FUNCTION "ASCF_GetVDIntOutputList" : Word
{ S7_Optimized_Access := 'TRUE' }
VERSION : 0.1
   VAR_INPUT
      Index : UInt;
   END_VAR

   VAR_OUTPUT
      QC : Byte;
      Value : DInt;
   END_VAR

   VAR_IN_OUT
      Outputs : Array[*] of "ASCF_CL_OutputType";
   END_VAR

   VAR_TEMP
      tempLowerBound : DInt;
      tempUpperBound : DInt;
      tempResult : Word;
      tempUnionType : "ASCF_UnionType";
      constErrors : "ASCF_CL_EnumErrors";
      constUnionTypes : "ASCF_EnumUnionTypes";
   END_VAR


BEGIN
	#tempResult := "ASCF_GetValueOutputList"(Index := #Index, Value => #tempUnionType, Outputs := #Outputs);

	IF #tempResult <> #constErrors.None THEN
	    #ASCF_GetVDIntOutputList := #tempResult;
	    RETURN;
	END_IF;

	IF #tempUnionType.Typeselector <> #constUnionTypes.VDInt THEN
	    #ASCF_GetVDIntOutputList := #constErrors.TypesDoNotMatch;
	    RETURN;
	END_IF;

	#QC := #tempUnionType.VQC;
	#Value := #tempUnionType.VDInt;
	#ASCF_GetVDIntOutputList := #constErrors.None;
END_FUNCTION